(* IEC 61131-3 sources: SRCI/RobotLibrary/Library/Interfaces, 2 files *)

(* ---- IMessageLogger.st ---- *)
INTERFACE IMessageLogger

METHOD PUBLIC AddMessageLog
VAR_INPUT
  /// Message to add to the log
  MessageLog : AlarmMessage;
END_VAR

END_METHOD

METHOD PUBLIC AddSystemLog
VAR_INPUT
  /// System messafe to add to the log
  SystemLog : STRING(RobotLibraryParameter.MESSAGE_TEXT_LEN);
END_VAR

END_METHOD

(* ---- IRobotLibraryCommandFB.st ---- *)
INTERFACE IRobotLibraryCommandFB

METHOD PUBLIC CallBack : DINT
VAR_INPUT
  /// Response data
  RspData : AxesGroupAcyclicAcrEntryRspBuffer;
END_VAR

END_METHOD

PROPERTY CommandData : RobotLibrarySendDataFB

GET

END_GET

SET

END_SET
